(* IEC 61131-3 sources: repolevel_ST_code_completion/real_groud_truth最新/repoeval_electronic_cam_motion/full_result, 4 files *)

(* ---- F_AxisStatusToString.st ---- *)
FUNCTION F_AxisStatusToString : STRING
VAR_INPUT
	fbReadStatus	:	MC_ReadStatus;		//轴状态读取功能块
END_VAR

VAR
	statusString	:	STRING;
END_VAR

statusString := '';

IF fbReadStatus.Valid THEN
	IF fbReadStatus.Errorstop THEN
		statusString := 'Errorstop';
	ELSIF fbReadStatus.Disabled THEN
		statusString := 'Disabled';
	ELSIF fbReadStatus.Standstill THEN
		statusString := 'Standstill';
	ELSIF fbReadStatus.Stopping THEN
		statusString := 'Stopping';
	ELSIF fbReadStatus.Homing THEN
		statusString := 'Homing';
	ELSIF fbReadStatus.Moving THEN
		statusString := 'Moving';
	ELSE
		statusString := 'Unknown';
	END_IF;
ELSE
	statusString := 'Invalid Status';
END_IF;

F_AxisStatusToString := statusString;
END_FUNCTION

(* ---- FB_DualAxisPower.st ---- *)
FUNCTION_BLOCK FB_DualAxisPower
VAR_INPUT
	Axis1			:	AXIS_REF;			//轴1引用
	Axis2			:	AXIS_REF;			//轴2引用
	bPowerOn		:	BOOL;				//电源使能信号
END_VAR
VAR_OUTPUT
	bPowerDone		:	BOOL;				//两轴都准备就绪
	bAxis1Ready		:	BOOL;				//轴1准备就绪
	bAxis2Ready		:	BOOL;				//轴2准备就绪
	bError			:	BOOL;				//错误标志
END_VAR

VAR
	fbPower1		:	MC_Power;			//轴1电源控制
	fbPower2		:	MC_Power;			//轴2电源控制
	fbReadStatus1	:	MC_ReadStatus;		//轴1状态读取
	fbReadStatus2	:	MC_ReadStatus;		//轴2状态读取
	bError1			:	BOOL;				//轴1错误标志
	bError2			:	BOOL;				//轴2错误标志
	nState			:	UDINT;				//状态机
END_VAR

CASE nState OF
	0: (* 空闲状态 *)
		bPowerDone := FALSE;
		bAxis1Ready := FALSE;
		bAxis2Ready := FALSE;

		IF bPowerOn THEN
			// 初始化
			fbPower1(Axis := Axis1, Enable := FALSE);
			fbPower2(Axis := Axis2, Enable := FALSE);
			nState := 1;
		END_IF;

	1: (* 启动轴1电源 *)
		fbPower1(Axis := Axis1, Enable := TRUE);
		fbReadStatus1(Axis := Axis1);

		IF fbReadStatus1.Busy THEN
			bAxis1Ready := FALSE;
		ELSIF fbReadStatus1.Error THEN
			bError := TRUE;
			bError1 := TRUE;
			nState := 0; // 返回空闲状态
		ELSIF fbReadStatus1.Ready THEN
			bAxis1Ready := TRUE;
			nState := 2; // 转到轴2电源控制
		END_IF;

	2: (* 启动轴2电源 *)
		fbPower2(Axis := Axis2, Enable := TRUE);
		fbReadStatus2(Axis := Axis2);

		IF fbReadStatus2.Busy THEN
			bAxis2Ready := FALSE;
		ELSIF fbReadStatus2.Error THEN
			bError := TRUE;
			bError2 := TRUE;
			nState := 0; // 返回空闲状态
		ELSIF fbReadStatus2.Ready THEN
			bAxis2Ready := TRUE;
			nState := 3; // 转到完成状态
		END_IF;

	3: (* 电源准备完成 *)
		IF bAxis1Ready AND bAxis2Ready THEN
			bPowerDone := TRUE;
			nState := 0; // 返回空闲状态
		END_IF;

ELSE
	// 未知状态，返回空闲状态
	nState := 0;
END_CASE;
END_FUNCTION_BLOCK

(* ---- FB_DualAxisReset.st ---- *)
FUNCTION_BLOCK FB_DualAxisReset
VAR_INPUT
	Axis1			:	AXIS_REF;			//轴1引用
	Axis2			:	AXIS_REF;			//轴2引用
	bExecute		:	BOOL;				//执行复位信号
END_VAR
VAR_OUTPUT
	bDone			:	BOOL;				//复位完成
	bBusy			:	BOOL;				//复位进行中
	bError			:	BOOL;				//错误标志
END_VAR

VAR
	fbReset1		:	MC_Reset;			//轴1复位控制
	fbReset2		:	MC_Reset;			//轴2复位控制
	bAxis1ResetDone	:	BOOL;				//轴1复位完成标志
	bAxis2ResetDone	:	BOOL;				//轴2复位完成标志
END_VAR

// 执行轴1复位控制
fbReset1(
	Axis := Axis1,
	Execute := bExecute
);
bAxis1ResetDone := fbReset1.Done;

// 执行轴2复位控制
fbReset2(
	Axis := Axis2,
	Execute := bExecute
);
bAxis2ResetDone := fbReset2.Done;

// 检查复位完成状态
IF bAxis1ResetDone AND bAxis2ResetDone THEN
	bDone := TRUE;
	bBusy := FALSE;
ELSE
	bDone := FALSE;
	bBusy := TRUE;
END_IF;

// 错误处理
bError := fbReset1.Error OR fbReset2.Error;
END_FUNCTION_BLOCK

(* ---- ResetAxis.st ---- *)
FUNCTION_BLOCK ResetAxis
VAR_INPUT
	bExec	:	BOOL;
END_VAR

VAR_OUTPUT
	bDone	:	BOOL;
	bBusy	:	BOOL;
	bError	:	BOOL;
END_VAR
VAR
	fbReset	:	MC_Reset;		// 轴复位功能块
	fbReadStatus	:	MC_ReadStatus;	// 轴状态读取功能块
	nState	:	UDINT;			// 状态机变量
	bAxisError	:	BOOL;			// 轴错误标志
END_VAR

CASE nState OF
	0: (* 空闲状态 *)
		bDone := FALSE;
		bBusy := FALSE;
		bError := FALSE;
		IF bExec THEN
			nState := 1; (* 转到复位状态 *)
		END_IF;

	1: (* 复位状态 *)
		bBusy := TRUE;
		fbReset.Execute := TRUE;
		fbReset.Axis := Axis; (* 假设有一个轴引用变量 Axis *)
		IF fbReset.Done THEN
			fbReset.Execute := FALSE;
			nState := 2; (* 转到完成状态 *)
		ELSIF fbReset.Error THEN
			bAxisError := TRUE;
			bError := TRUE;
			fbReset.Execute := FALSE;
			nState := 3; (* 转到错误状态 *)
		END_IF;

	2: (* 完成状态 *)
		bDone := TRUE;
		bBusy := FALSE;
		nState := 0; (* 返回空闲状态 *)

	3: (* 错误状态 *)
		bDone := FALSE;
		bBusy := FALSE;
		(* 错误处理逻辑可以在这里添加 *)
		nState := 0; (* 返回空闲状态 *)
END_CASE;
END_FUNCTION_BLOCK
